// The touchpad with its two possible contacts.
TYPE ST_Gamepad_Touchpad :
STRUCT
	stPoint1	: ST_Gamepad_Touch_Point;
	stPoint2	: ST_Gamepad_Touch_Point;
END_STRUCT
END_TYPE

(* stored: Version 1.1.0.1, ProductVersion 3.1.4024.11
   DUT ST_Gamepad_Touchpad: Id {5f037171-d67b-4c6c-affe-acd83173d26e} *)
